FUNCTION_BLOCK fbAbsolute
VAR_INPUT
	boEnable	:BOOL;
	boStart		:BOOL;
	
	lrPos		:LREAL;
	lrVelo		:LREAL;
	lrAcc		:LREAL;
	lrDec		:LREAL;
	lrJerk		:LREAL;
END_VAR
VAR_OUTPUT
END_VAR
VAR
	iState		:INT:=0;
	sState		:STRING;
	rtrboStart	:R_trig;
	ftrboEnable	:f_trig;
	tonMoveNotDone	:ton;
END_VAR
VAR_IN_OUT
	fbPower		:mc_Power;
	fbAbsolute  :mc_MoveAbsolute;
	axis		:axis_ref;
END_VAR


rtrboStart(CLK:=boStart);
ftrboEnable(CLK:=boEnable);

CASE iState OF
0:
	IF boEnable THEN
		iState:=100;
	END_IF
100:
	IF rtrboStart.Q THEN
		fbAbsolute.Execute:=TRUE;
		tonMoveNotDone.IN:=TRUE;
		iState:=1000;
	END_IF
1000:
	fbAbsolute.Execute:=FALSE;
	IF fbAbsolute.Done  THEN
		tonMoveNotDone.IN:=FALSE;
		iState:=100;
	ELSIF tonMoveNotDone.Q THEN
		sState:='motor dont have achived target position';
		tonMoveNotDone.IN:=FALSE;
		iState:=100;
	END_IF	
END_CASE

tonMoveNotDone(PT:=T#100s);

IF ftrboEnable.Q THEN
	iState:=0;
	sState:='';
	fbAbsolute.Execute:=FALSE;
	tonMoveNotDone.IN:=FALSE;
END_IF

fbPower(
	Axis:=axis , 
	Enable:=boEnable , 
	Enable_Positive:=boEnable , 
	Enable_Negative:=boEnable , 
	Override:=100);
	
fbAbsolute(
	Axis:=axis , 
	Position:=lrPos , 
	Velocity:=lrVelo , 
	Acceleration:=lrAcc , 
	Deceleration:=lrDec , 
	Jerk:=lrJerk  );

END_FUNCTION_BLOCK

(* stored: Version 1.1.0.1, ProductVersion 3.1.4024.12
   POU fbAbsolute: Id {73cc4ffd-d83d-468f-8f36-2038d1eb11a3}, SpecialFunc None *)
